(* CoDeSys 2.3 library: SysLibVisu.lib *)

(* Data type *)
TYPE VisualObjectType
STRUCT
	(* Absolut movement *)
 	nXOffset:INT;
  	nYOffset:INT;
	nScale:INT;
	nAngle:INT;

	(* Variables *)
	bInvisible:BOOL;
	stTextDisplay:STRING;
	bToggleColor:BOOL;
	bInputDisabled: BOOL;
	stTooltipDisplay:STRING;

	(* Text and font *)
  	dwTextFlags:DWORD;
	dwTextColor:DWORD;
	nFontHeight:INT;
	dwFontFlags:DWORD;
	stFontName:STRING;

	(* Line *)
	nLineWidth:INT;

	(* Color *)
	dwFillColor: DWORD;
	dwFillColorAlarm: DWORD;
	dwFrameColor: DWORD;
	dwFrameColorAlarm: DWORD;
	dwFillFlags: DWORD;
	dwFrameFlags: DWORD;

	(* Relative movement *)
	nLeft:INT;
	nTop:INT;
	nRight:INT;
	nBottom:INT;
END_STRUCT
END_TYPE
